// TIA Portal V17 export
// export: Created 2023-04-11T09:33:25.1860708Z, ExportSetting WithDefaults, DisplayName Totally Integrated Automation Portal, DisplayVersion V17 Update 3, DisplayName TIA Portal Openness, DisplayVersion V17 Update 3, DisplayName TIA Portal Version Control Interface, DisplayVersion V17, DisplayName SINAMICS Startdrive Advanced, DisplayVersion V17 Update2, DisplayName SINAMICS Startdrive G130, G150, S120, S150, SINAMICS MV, S210, DisplayVersion V17 Update2, DisplayName SINAMICS Startdrive G110M, G120, G120C, G120D, G120P, G115D, DisplayVersion V17 Update2, DisplayName STEP 7 Professional, DisplayVersion V17 Update 3, DisplayName STEP 7 Safety, DisplayVersion V17, DisplayName WinCC UA Professional, DisplayVersion V17 Update 3
FUNCTION_BLOCK "FB_stdStepStart"   // FB17, LAD
{ S7_Optimized_Access := 'TRUE' }
VERSION : 0.1
// Standard program step
// stored: AutoNumber true, IsIECCheckEnabled false, IsRetainMemResEnabled false, MemoryReserve 100, SetENOAutomatically false, UDAEnableTagReadback false
   VAR_INPUT
      enable { ExternalAccessible := 'False'; ExternalVisible := 'False'; ExternalWritable := 'False'} : Bool;
      allow : Bool;
      condition { ExternalAccessible := 'False'; ExternalVisible := 'False'; ExternalWritable := 'False'} : Bool;
      trigger : Bool;
      delay { ExternalAccessible := 'False'; ExternalVisible := 'False'; ExternalWritable := 'False'} : Time;
      errTime { ExternalAccessible := 'False'; ExternalVisible := 'False'; ExternalWritable := 'False'} : Time;
   END_VAR
   VAR_OUTPUT
      done { ExternalAccessible := 'False'; ExternalVisible := 'False'; ExternalWritable := 'False'} : Bool;
      error { ExternalAccessible := 'False'; ExternalVisible := 'False'; ExternalWritable := 'False'} : Bool;
   END_VAR
   VAR
      temp_1 { ExternalAccessible := 'False'; ExternalVisible := 'False'; ExternalWritable := 'False'} : Bool;
      temp_2 { ExternalAccessible := 'False'; ExternalVisible := 'False'; ExternalWritable := 'False'} : Bool;
      IEC_Timer_Instance_1 { ExternalAccessible := 'False'; ExternalVisible := 'False'; ExternalWritable := 'False'; S7_SetPoint := 'True'} : TON_TIME;
      IEC_Timer_0_Instance { S7_SetPoint := 'True'} : TP_TIME;
   END_VAR
BEGIN

REGION Network 1: Done and Error output logic
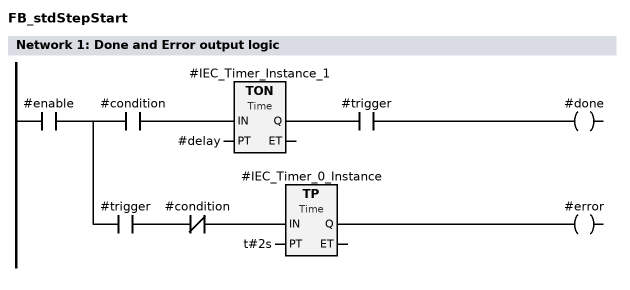
   RUNG wire#powerrail
      Contact( #enable )
      wire#w1
      Contact( #condition )
      { S7_Templates := "time_type := Time" } #IEC_Timer_Instance_1.TON(pt := #delay, et =>)
      Contact( #trigger )
      Coil( #done )
   END_RUNG
   RUNG wire#w1
      Contact( #trigger )
      I_Contact( #condition )
      { S7_Templates := "time_type := Time" } #IEC_Timer_0_Instance.TP(pt := t#2s, et =>)
      Coil( #error )
   END_RUNG
   // the same network as SCL:
   #IEC_Timer_Instance_1(IN := #enable AND #condition, PT := #delay);   // TON
   #done := #IEC_Timer_Instance_1.Q AND #trigger;
   #IEC_Timer_0_Instance(IN := #enable AND #trigger AND NOT #condition, PT := t#2s);   // TP
   #error := #IEC_Timer_0_Instance.Q;
END_REGION
END_FUNCTION_BLOCK
